(* CoDeSys 2.3 export: FK16PUMPAUTOCONTROL.EXP *)

(* POU K16/fK16PumpAutoControl, ST *)
FUNCTION fK16PumpAutoControl : BOOL
VAR_INPUT
	PumpID : USINT;
	EmergencyPumpStopButtonPressed : BOOL;
END_VAR
IF EmergencyPumpStopButtonPressed THEN	(*Нажат аварийный стоп насоса?*)
	fTurnOffK16Pump(PumpID); (*Выключить насос*)
	RETURN;
END_IF;

IF K16PumpFaulty[PumpID] THEN
	fTurnOffK16Pump(PumpID); (*Выключить насос*)
ELSE
	fTurnOnK16Pump(PumpID); (*Включить насос*)
END_IF;
END_FUNCTION
